FUNCTION F_ConfigCommunicationEmulation : BOOL

;

END_FUNCTION

(* stored: Version 1.1.0.1, ProductVersion 3.1.4024.9
   POU F_ConfigCommunicationEmulation: Id {d700ac22-5cfb-4b93-816e-bb60783ad3fa}, SpecialFunc None *)
